FUNCTION_BLOCK ABSTRACT CollectionEventHandler EXTENDS CollectionEventHandlerBase
VAR
	expectedOriginator : I_Collection;
END_VAR

METHOD FB_init : BOOL
VAR_INPUT
	bInitRetains : BOOL; // if TRUE, the retain variables are initialized (warm start / cold start)
	bInCopyCode : BOOL;  // if TRUE, the instance afterwards gets moved into the copy code (online change)
	ExpectedOriginator : I_Collection;
END_VAR
SetExpectedOriginator(ExpectedOriginator);
END_METHOD

METHOD PUBLIC SetExpectedOriginator
VAR_INPUT
	ExpectedOriginator : I_Collection;
END_VAR
THIS^.expectedOriginator := ExpectedOriginator;
END_METHOD

END_FUNCTION_BLOCK

(* stored: Version 1.1.0.1, ProductVersion 3.1.4024.12
   POU CollectionEventHandler: Id {b4addd9b-b561-0d3c-0b54-65e515323951}, SpecialFunc None
   Folder Constructor: Id {59b859c2-f83b-0e38-2144-4867755b0805}
   Method FB_init: Id {c9bc5149-35be-0e55-3328-c406d13d81eb}
   Method SetExpectedOriginator: Id {9d6f43ab-bd55-0f0b-0e65-e1dc52ed0f0c} *)
